FUNCTION "Proc_Lanc_Fab" : String
{ S7_Optimized_Access := 'TRUE' }
VERSION : 0.1
   VAR_OUTPUT
      Msg_Def : String;
      Err_Sql : String;
   END_VAR

   VAR_IN_OUT
      Data_Dosage : "S_Suivi_Dosage";
   END_VAR

   VAR_TEMP
      parameters_value : Array[0..20] of String;
      Resultat_Decode : WString[4000];
      status : Int;
   END_VAR


BEGIN
	//Insertion des parametres
	#parameters_value[0] := UINT_TO_STRING("Num_Poste");
	#parameters_value[1] := ULINT_TO_STRING(#Data_Dosage._IdHDos);

	//++++++++++++++++++++++++++++++++++++++++++++++++++++++++++++++++++++++++++++++//

	#Resultat_Decode := "COMBASE"(procedure_name := 'SP_Dos_LancFab',
	                              values_of_record := #parameters_value,
	                              parameters_number := 2,
	                              ERROR_MESSAGE => #Err_Sql);

	//++++++++++++++++++++++++++++++++++++++++++++++++++++++++++++++++++++++++++++++//

	#status := "FCT_DECODE_TRAME"(KEYWORD := 'REPONSE:',
	                              BUFFER := #Resultat_Decode,
	                              Retour_VAL => #Proc_Lanc_Fab);

	IF #Proc_Lanc_Fab = 'NOK' THEN
	    #status := "FCT_DECODE_TRAME"(KEYWORD := 'MESS:',
	                                  BUFFER := #Resultat_Decode,
	                                  Retour_VAL => #Msg_Def);
	    RETURN;
	ELSIF #Proc_Lanc_Fab = 'OK' THEN
	    #status := "FCT_DECODE_TRAME"(KEYWORD := 'MESS:',
	                                  BUFFER := #Resultat_Decode,
	                                  Retour_VAL => #Msg_Def);
	    IF #Msg_Def = 'VIDE' THEN
	        RETURN;
	    END_IF;
	ELSE
	    RETURN;
	END_IF;
END_FUNCTION

